% RSLogix 500 project SEND_DATA_BAK068.RSS, saved by version 8.10.00.18 %
PROJECT "UNTITLED"    % processor: Bul.1763 MicroLogix 1100 Series B %

PROGRAM FILES
  LAD 2 "MAIN"  2 rungs
  LAD 3 "CLOCK"  14 rungs
  LAD 4   12 rungs

DATA FILES
  O0 OUTPUT  4 elements
  I1 INPUT  6 elements
  S2 STATUS  66 elements
  B3 BINARY  1 elements
  T4 TIMER  4 elements
  C5 COUNTER  2 elements
  R6 CONTROL  1 elements
  N7 INTEGER  11 elements
  F8 FLOAT  1 elements

LADDER 2 "MAIN"
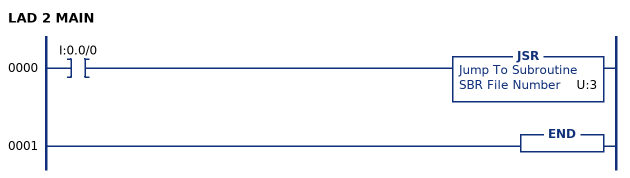
% Rung: 0 %
SOR XIC I:0.0/0 JSR U:3 EOR
%   XIC I:0.0/0  "send_data" %
% Rung: 1 %
SOR END EOR

LADDER 3 "CLOCK"
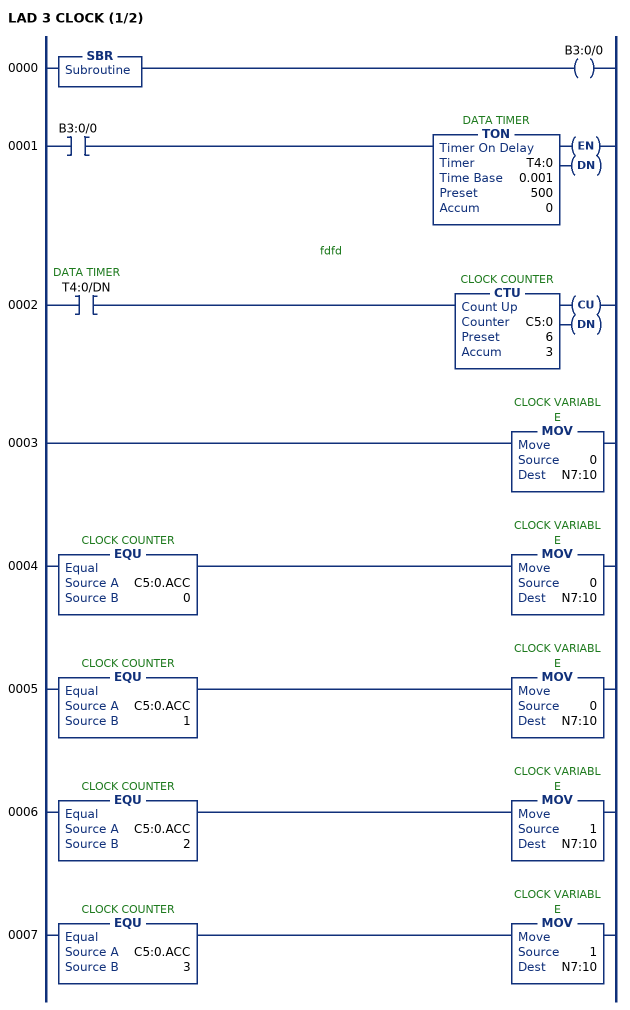
% Rung: 0 %
SOR SBR OTE B3:0/0 EOR
% Rung: 1 %
SOR XIC B3:0/0 TON T4:0 0.001 500 0 EOR
%   T4:0  "DATA TIMER" %
% Rung: 2 %
% fdfd %
SOR XIC T4:0/DN CTU C5:0 6 3 EOR
%   T4:0  "DATA TIMER" %
%   C5:0  "CLOCK COUNTER" %
% Rung: 3 %
SOR MOV 0 N7:10 EOR
%   N7:10  "CLOCK VARIABLE" %
% Rung: 4 %
SOR EQU C5:0.ACC 0 MOV 0 N7:10 EOR
%   C5:0  "CLOCK COUNTER" %
%   N7:10  "CLOCK VARIABLE" %
% Rung: 5 %
SOR EQU C5:0.ACC 1 MOV 0 N7:10 EOR
%   C5:0  "CLOCK COUNTER" %
%   N7:10  "CLOCK VARIABLE" %
% Rung: 6 %
SOR EQU C5:0.ACC 2 MOV 1 N7:10 EOR
%   C5:0  "CLOCK COUNTER" %
%   N7:10  "CLOCK VARIABLE" %
% Rung: 7 %
SOR EQU C5:0.ACC 3 MOV 1 N7:10 EOR
%   C5:0  "CLOCK COUNTER" %
%   N7:10  "CLOCK VARIABLE" %

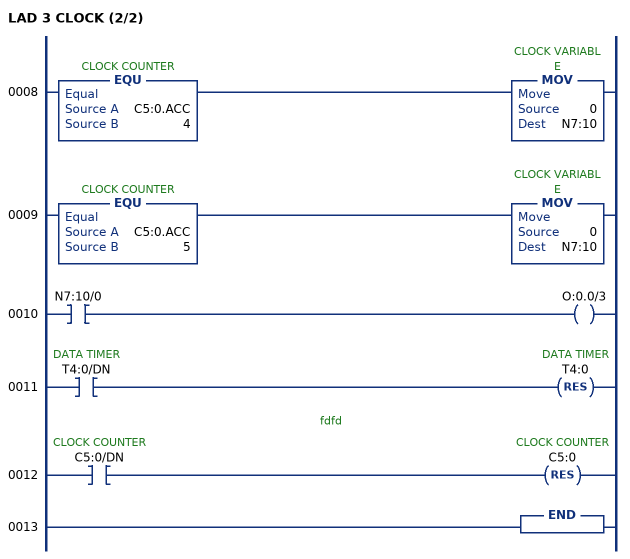
% Rung: 8 %
SOR EQU C5:0.ACC 4 MOV 0 N7:10 EOR
%   C5:0  "CLOCK COUNTER" %
%   N7:10  "CLOCK VARIABLE" %
% Rung: 9 %
SOR EQU C5:0.ACC 5 MOV 0 N7:10 EOR
%   C5:0  "CLOCK COUNTER" %
%   N7:10  "CLOCK VARIABLE" %
% Rung: 10 %
SOR XIC N7:10/0 OTE O:0.0/3 EOR
% Rung: 11 %
SOR XIC T4:0/DN RES T4:0 EOR
%   T4:0  "DATA TIMER" %
% Rung: 12 %
% fdfd %
SOR XIC C5:0/DN RES C5:0 EOR
%   C5:0  "CLOCK COUNTER" %
% Rung: 13 %
SOR END EOR

LADDER 4
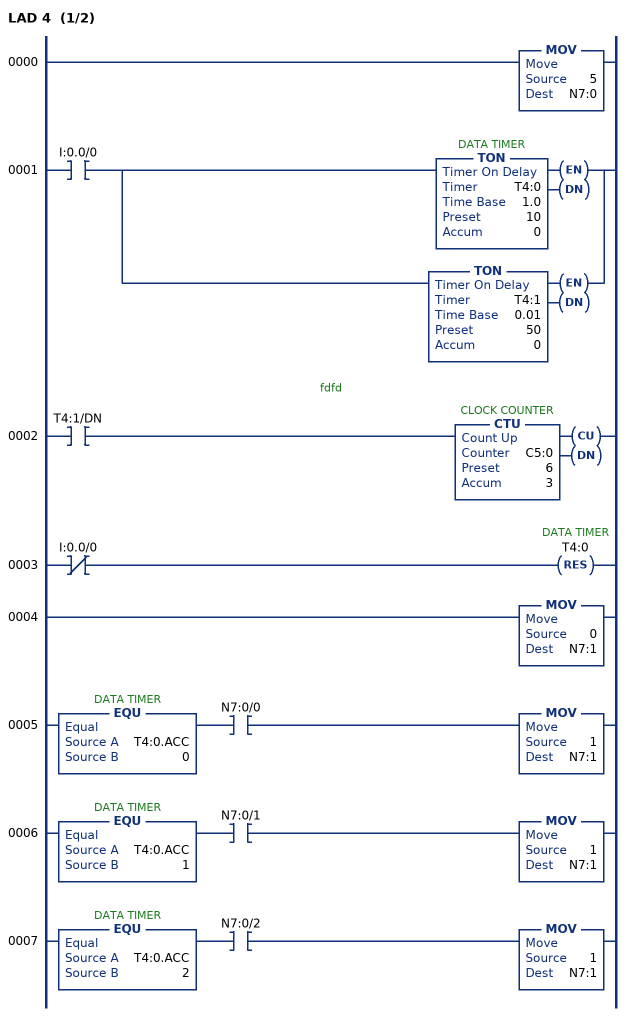
% Rung: 0 %
SOR MOV 5 N7:0 EOR
% Rung: 1 %
SOR XIC I:0.0/0 BST TON T4:0 1.0 10 0 NXB TON T4:1 0.01 50 0 BND EOR
%   XIC I:0.0/0  "send_data" %
%   T4:0  "DATA TIMER" %
%   TON T4:1  "DATA TIMER" %
% Rung: 2 %
% fdfd %
SOR XIC T4:1/DN CTU C5:0 6 3 EOR
%   XIC T4:1/DN  "timer_reached" %
%   C5:0  "CLOCK COUNTER" %
% Rung: 3 %
SOR XIO I:0.0/0 RES T4:0 EOR
%   T4:0  "DATA TIMER" %
% Rung: 4 %
SOR MOV 0 N7:1 EOR
% Rung: 5 %
SOR EQU T4:0.ACC 0 XIC N7:0/0 MOV 1 N7:1 EOR
%   T4:0  "DATA TIMER" %
% Rung: 6 %
SOR EQU T4:0.ACC 1 XIC N7:0/1 MOV 1 N7:1 EOR
%   T4:0  "DATA TIMER" %
% Rung: 7 %
SOR EQU T4:0.ACC 2 XIC N7:0/2 MOV 1 N7:1 EOR
%   T4:0  "DATA TIMER" %

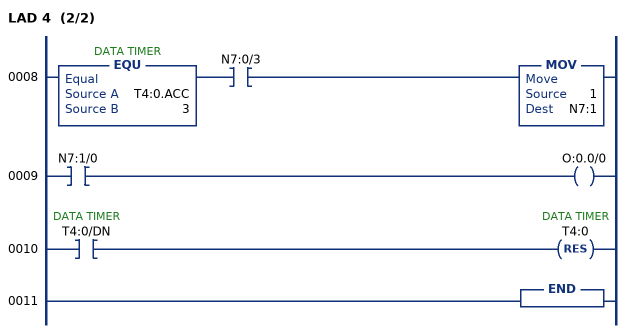
% Rung: 8 %
SOR EQU T4:0.ACC 3 XIC N7:0/3 MOV 1 N7:1 EOR
%   T4:0  "DATA TIMER" %
% Rung: 9 %
SOR XIC N7:1/0 OTE O:0.0/0 EOR
% Rung: 10 %
SOR XIC T4:0/DN RES T4:0 EOR
%   T4:0  "DATA TIMER" %
% Rung: 11 %
SOR END EOR

OTHER DOCUMENTED ADDRESSES
  O:0.0/1  "SCL"
  U3  

DATA TABLE (non-zero values as saved)
DATA T4
% .PRE .ACC %
% T4:0 % 500 0
% T4:1 % 50 0
% T4:2 % 10 0
% T4:3 % 10 0
DATA C5
% .PRE .ACC %
% C5:0 % 6 3
% C5:1 % 4 0
DATA N7
% N7:0 % 3 1 0 0 0 0 0 0 0 0
